PROGRAM POU_Test
VAR
	fbDirectoryContorlTest : FB_DirectoryContorlTest;
END_VAR

//TcUnit.RUN();

END_PROGRAM

(* stored: Version 1.1.0.1, ProductVersion 3.1.4024.12
   POU POU_Test: Id {6076125f-0f1a-40bc-9da2-35429578d6d9}, SpecialFunc None *)
